// VisionSensors/Balluff BVS/fbBvsControl_ComIO
FUNCTION_BLOCK fbBvsControl_ComIO IMPLEMENTS I_VisionSensorSTD
VAR_IN_OUT
	stIO_Data: stVisionSensor_DigInOut;
END_VAR
VAR_INPUT
	bTrigger:BOOL;
	bReadActualInspection:BOOL;
	bChangeInspection:BOOL;		// Zbocze narastające inicjuje zmianę programu
	iInspectionToActive:INT;
	tMinImpWidth:TIME;		// Czas minimalnego trwania impulsu
END_VAR
VAR_OUTPUT
	bBusy: BOOL;
	bOutput1: BOOL;
	bOutput2: BOOL;
	bOutput3: BOOL;
	bError:	BOOL;
	bResultReady: BOOL;
	iActiveProgramId:INT;
END_VAR
VAR
	iWorkStep:INT;
	fbTP_ImpuleGen:TP;
	iImpulseToGenerate:INT;
	wConfirmedDeterctionNumber: WORD;
	fbTON_NewImpulsePause: TON;
	fbTON_Timeout: TON;
	bToggleMemory: BOOL;
	bNewInspectionBusy :BOOL;
	fbTON_CmdTimeout: TON;
	bReadInspectionBusy: BOOL;
	bSetInspectionBusy: BOOL;
	iIdToSet: INT;
	fbTON_NewStep: TON;
	fbTP_ImpulesRead: TP;
	fbTON_NewStepLong: TON;
	iTargetIdToSet: INT;
END_VAR

IF iWorkStep > 10 THEN
	fbTP_ImpuleGen(IN:= FALSE, PT:= tMinImpWidth + T#5MS);	
	fbTP_ImpulesRead(IN:= FALSE, PT:= 2*tMinImpWidth);	
	fbTON_NewStep(IN:= TRUE,PT:= tMinImpWidth);
	fbTON_NewStepLong(IN:= TRUE,PT:= 2*tMinImpWidth);
	IF iWorkStep < 90 THEN
		fbTON_CmdTimeout(IN:= TRUE, PT:= T#7S);
		IF fbTON_CmdTimeout.Q THEN
			fbTON_CmdTimeout(IN:= FALSE);
			iWorkStep := 90;
		END_IF
	END_IF	
END_IF


CASE iWorkStep OF
	0:	// Inicjalizacja
		IF bNewInspectionBusy OR bTrigger THEN		// Nowa detekcja
			bBusy := TRUE;
			bError := bSetInspectionBusy := bReadInspectionBusy := bOutput1 := bOutput2 := bOutput3 := bResultReady := FALSE;
			stIO_Data.bOut0_Trigger := TRUE;
			bToggleMemory:= stIO_Data.bIn0;
			fbTON_CmdTimeout(IN:= FALSE);
			iWorkStep := 10;
		ELSIF bReadInspectionBusy OR bReadActualInspection THEN		// Odczyt Id detekcji
			bBusy := TRUE;
			bError := bSetInspectionBusy := bResultReady := FALSE;
			iIdToSet := 21;
			iActiveProgramId := -1;
			fbTON_CmdTimeout(IN:= FALSE);
			iWorkStep := 20;
		ELSIF bSetInspectionBusy OR bChangeInspection THEN			// Ustawienie nowej detekcji
			IF bChangeInspection THEN
				IF iInspectionToActive > 0 AND iInspectionToActive <= 20 THEN
					iIdToSet := iInspectionToActive;
				END_IF		
			END_IF
			IF iIdToSet > 0 AND iIdToSet <= 20 THEN 			
				bBusy := TRUE;
				bError := bResultReady := FALSE;
				iTargetIdToSet:= iIdToSet;
				iActiveProgramId := -1;
				fbTON_CmdTimeout(IN:= FALSE);
				iWorkStep := 20;
			ELSE	
				bBusy := FALSE;
				bError := bResultReady := TRUE;
				iActiveProgramId := -1;
				iWorkStep := 1;
			END_IF
		END_IF
		
	1:	// Oczekiwanie po wykonanej komendzie na sygnał zerowy na poszczególnych wejściach
		IF NOT bTrigger AND NOT bReadActualInspection AND NOT bChangeInspection THEN
			fbTON_CmdTimeout(IN:= TRUE, PT:= T#1S);
			IF (NOT bNewInspectionBusy AND NOT bReadInspectionBusy AND NOT bSetInspectionBusy) OR fbTON_CmdTimeout.Q THEN
				bNewInspectionBusy := bReadInspectionBusy := bSetInspectionBusy := FALSE;
				bBusy := stIO_Data.bOut0_Trigger := stIO_Data.bOut1 := FALSE;
				fbTON_CmdTimeout(IN:= FALSE);
				iWorkStep := 0;
			END_IF	
		END_IF
	
	10:	// Detekcja wyzwolona, oczekiwanie na rezultat
		fbTON_CmdTimeout(IN:= TRUE, PT:= T#500MS);
		IF bToggleMemory <> stIO_Data.bIn0 THEN		// Detekcja zakończona
			bOutput1 := stIO_Data.bIn1;
			bOutput2 := stIO_Data.bInOut2;
			bOutput3 := stIO_Data.bInOut3;
			bResultReady := TRUE;
			bBusy := FALSE;
			bToggleMemory := stIO_Data.bIn0;
			stIO_Data.bOut0_Trigger := FALSE;
			iWorkStep := 1;
		ELSIF fbTON_CmdTimeout.Q THEN
			bBusy := FALSE;
			bError := TRUE;
			fbTON_CmdTimeout(IN:= FALSE);
			stIO_Data.bOut0_Trigger := FALSE;
			iWorkStep := 1;
		END_IF
		IF iWorkStep <> 10 THEN fbTON_CmdTimeout(IN:= FALSE); END_IF
				
		
	20:	// Odczyt/zmiana aktywnego programu 
		stIO_Data.bOut0_Trigger := stIO_Data.bOut1 := FALSE;
		fbTON_NewStep(IN:= FALSE);
		iWorkStep := 21;
	21:	// ***** FAZA 1 ***** Ustawienie sygnału wyboru programu	
		IF fbTON_NewStep.Q THEN
			stIO_Data.bOut1 := TRUE;
			fbTON_NewStep(IN:= FALSE);
			iWorkStep := 22;
		END_IF	
	22:	// ***** FAZA 2 ***** Oczekiwanie na wygaszenie wyjść i generacja impulsu
		IF NOT stIO_Data.bIn1 AND NOT stIO_Data.bInOut2 AND NOT stIO_Data.bInOut3 AND fbTON_NewStep.Q THEN
			fbTP_ImpuleGen(IN:= NOT stIO_Data.bOut0_Trigger);
			stIO_Data.bOut0_Trigger := fbTP_ImpuleGen.Q;
			iWorkStep := 23;	
		END_IF
	23:
		stIO_Data.bOut0_Trigger := fbTP_ImpuleGen.Q;
		IF NOT stIO_Data.bOut0_Trigger THEN
			fbTON_NewStep(IN:= FALSE);
			iWorkStep := 24;	
		END_IF	
	24:	// ***** FAZA 3 ***** Oczekiwanie na wystawienie wyjść
		IF stIO_Data.bIn1 AND stIO_Data.bInOut2 AND stIO_Data.bInOut3 AND fbTON_NewStep.Q THEN
			fbTON_NewStep(IN:= FALSE);
			iWorkStep := 25;	
		END_IF
	25:	// ***** FAZA 3 ***** Generacja liczby impulsów odpowiadających numerowi detekcji
		IF iIdToSet > 0 THEN
			iWorkStep := 26;
		ELSE
			fbTON_NewStep(IN:= FALSE);
			iWorkStep := 27;
		END_IF
	26:	// ***** FAZA 3 ***** Generacja liczby impulsów odpowiadających numerowi detekcji
		fbTP_ImpuleGen(IN:= NOT stIO_Data.bOut0_Trigger);
		stIO_Data.bOut0_Trigger := fbTP_ImpuleGen.Q;
		IF NOT stIO_Data.bOut0_Trigger THEN
			iIdToSet := iIdToSet -1;
			fbTON_NewStep(IN:= FALSE);
			iWorkStep := 27;
		END_IF
	27:	// ***** FAZA 3 ***** Pauza pomiędzy impulsami
		IF fbTON_NewStep.Q THEN
			IF iIdToSet > 0 THEN
				iWorkStep := 25;
			ELSE
				iWorkStep := 28;
			END_IF
		END_IF
	28:	// ***** FAZA 4 ***** Kasowanie sygnału ustawienia inspekcji
		stIO_Data.bOut0_Trigger := stIO_Data.bOut1 := FALSE;
		IF NOT stIO_Data.bIn1 AND NOT stIO_Data.bInOut2 AND NOT stIO_Data.bInOut3 THEN
			fbTON_NewStep(IN:= FALSE);
			iWorkStep := 29;
		END_IF
	29:	// Wystawienie pierwszego sygnału trigger
		IF fbTON_NewStep.Q THEN
			fbTP_ImpulesRead(IN:= NOT stIO_Data.bOut0_Trigger);
			stIO_Data.bOut0_Trigger := fbTP_ImpulesRead.Q;
			IF NOT stIO_Data.bOut0_Trigger THEN
				wConfirmedDeterctionNumber.0 := stIO_Data.bIn1;
				wConfirmedDeterctionNumber.1 := stIO_Data.bInOut2;
				wConfirmedDeterctionNumber.2 := stIO_Data.bInOut3;
				fbTON_NewStepLong(IN:= FALSE);
				iWorkStep := 30;
			END_IF
		END_IF
		
	30:
		IF NOT stIO_Data.bIn1 AND NOT stIO_Data.bInOut2 AND NOT stIO_Data.bInOut3 AND fbTON_NewStepLong.Q THEN
			fbTON_NewStep(IN:= FALSE);
			iWorkStep := 31;
		END_IF
	31:
		IF fbTON_NewStep.Q THEN
			fbTP_ImpulesRead(IN:= NOT stIO_Data.bOut0_Trigger);
			stIO_Data.bOut0_Trigger := fbTP_ImpulesRead.Q;
			IF NOT stIO_Data.bOut0_Trigger THEN
				wConfirmedDeterctionNumber.3 := stIO_Data.bIn1;
				wConfirmedDeterctionNumber.4 := stIO_Data.bInOut2;
				wConfirmedDeterctionNumber.5 := stIO_Data.bInOut3;
				fbTON_NewStepLong(IN:= FALSE);
				iWorkStep := 32;
			END_IF
		END_IF
	32:
		IF NOT stIO_Data.bIn1 AND NOT stIO_Data.bInOut2 AND NOT stIO_Data.bInOut3 AND fbTON_NewStepLong.Q THEN
			fbTON_NewStep(IN:= FALSE);
			iWorkStep := 33;
		END_IF
	33:
		IF fbTON_NewStep.Q THEN
			fbTP_ImpuleGen(IN:= NOT stIO_Data.bOut0_Trigger);
			stIO_Data.bOut0_Trigger := fbTP_ImpuleGen.Q;
			IF NOT stIO_Data.bOut0_Trigger THEN
				iWorkStep := 34;
			END_IF
		END_IF
	34:
		IF NOT stIO_Data.bIn1 AND NOT stIO_Data.bInOut2 AND NOT stIO_Data.bInOut3 THEN
			bBusy := FALSE;
			iActiveProgramId := WORD_TO_INT(wConfirmedDeterctionNumber);
			bResultReady := TRUE;
			bError := iTargetIdToSet = iActiveProgramId;
			iWorkStep := 1;
		END_IF
			
	90:	// In case of error ...
		bError := TRUE;
		bBusy := FALSE;
		stIO_Data.bOut0_Trigger := stIO_Data.bOut1 := FALSE;
		fbTON_CmdTimeout(IN:= TRUE, PT:= T#2S);
		IF fbTON_CmdTimeout.Q THEN
			iWorkStep := 1; 
		END_IF

END_CASE

METHOD mNewInspection : BOOL (* Metoda zwraca true gdy detekcja zostanie zakończona*)
VAR_OUTPUT
	bError	: BOOL;			// Informacja zakończeniu detekcji z błędem
	bOut1, bOut2, bOut3, bOut4	: BOOL;		// Wyjścia zostają odświeżone po zakońcoznej detekcji 
END_VAR
IF iWorkStep = 0 THEN
	bOut1 := bOut2 := bOut3 := bOut1 := bResultReady := FALSE;
	bNewInspectionBusy := TRUE;
ELSIF bNewInspectionBusy THEN
	IF bResultReady THEN
		bOut1 := bOutput1;
		bOut2 := bOutput2;
		bOut3 := bOutput3;
		bNewInspectionBusy := bError := bOut4 := FALSE;
		mNewInspection := TRUE;
	ELSIF fbTON_CmdTimeout.Q THEN
		bError := mNewInspection := TRUE;	
		bNewInspectionBusy := FALSE;
	END_IF
ELSE
	bError := mNewInspection := TRUE;
END_IF
END_METHOD

METHOD mReadInspectionId : BOOL (* Metoda zwraca true gdy zakończyła pracę*)
VAR_OUTPUT
	bError	: BOOL;			// Błąd ustawienia
	iActiveInspectionId	: INT;		// Identyfikator aktualnej inspekcji
END_VAR
IF iWorkStep = 0 THEN
	bResultReady := FALSE;
	bReadInspectionBusy := TRUE;
ELSIF bReadInspectionBusy THEN
	IF bResultReady THEN
		bReadInspectionBusy := bError := FALSE;
		iActiveInspectionId := iActiveProgramId;
		mReadInspectionId := TRUE;
	ELSIF fbTON_CmdTimeout.Q THEN
		bError := mReadInspectionId := TRUE;	
		iActiveInspectionId := -1;
		bReadInspectionBusy := FALSE;
	END_IF
ELSE
	bError := mReadInspectionId := TRUE;
	iActiveInspectionId := -1;
END_IF
END_METHOD

METHOD mSetInspectionId : BOOL
VAR_OUTPUT
	bError	: BOOL; 		// Błąd ustawienia
	iActiveInspectionId	: INT;		// Identyfikator aktualnej inspekcji
END_VAR
VAR_INPUT
	iInspectionIdToSet	: INT;			// Identyfikator inspekcji do ustawienia
END_VAR
IF iWorkStep = 0 AND iInspectionIdToSet <= 20 AND iInspectionIdToSet > 0 THEN
	bResultReady := FALSE;
	iIdToSet := iInspectionIdToSet;
	bSetInspectionBusy := TRUE;
ELSIF bSetInspectionBusy THEN
	IF bResultReady THEN
		bSetInspectionBusy := bError := FALSE;
		bError := iActiveProgramId <> iInspectionIdToSet;
		iActiveInspectionId := iActiveProgramId;
		mSetInspectionId := TRUE;
	ELSIF fbTON_CmdTimeout.Q THEN
		bError := mSetInspectionId := TRUE;	
		iActiveInspectionId := -1;
		bSetInspectionBusy := FALSE;
	END_IF
ELSE
	bError := mSetInspectionId := TRUE;
	iActiveInspectionId := -1;
END_IF
END_METHOD

END_FUNCTION_BLOCK

// VisionSensors/Cognex/fbCognexIS280Control
FUNCTION_BLOCK fbCognexIS280Control IMPLEMENTS I_VisionSensorSTD
VAR_IN_OUT
	stIO_Data: stCognexIS280_DigInOut;
END_VAR
VAR_INPUT
	bTrigger:BOOL;
	bReadActualInspection:BOOL;
	bChangeInspection:BOOL;		// Zbocze narastające inicjuje zmianę programu
	iInspectionToActive:INT;
	tMinImpWidth:TIME;		// Czas minimalnego trwania impulsu
END_VAR
VAR_OUTPUT
	bBusy: BOOL;
	bOutput1: BOOL;
	bOutput2: BOOL;
	bOutput3: BOOL;
	bError:	BOOL;
	bResultReady: BOOL;
	iActiveProgramId:INT;
END_VAR
VAR
	iWorkStep:INT;
	fbTP_ImpuleGen:TP;
	fbTON_Timeout: TON;
	bNewInspectionBusy :BOOL;
	fbTON_CmdTimeout: TON;
	iIdToSet: INT;
	fbTON_NewStep: TON;
	fbTP_ImpulesRead: TP;
	fbTON_NewStepLong: TON;
	iTargetIdToSet: INT;
END_VAR


CASE iWorkStep OF
	0:	// Inicjalizacja
		IF bNewInspectionBusy OR bTrigger THEN		// Nowa detekcja
			bBusy := TRUE;
		//	bSetInspectionBusy := bReadInspectionBusy := FALSE;
			bError := bOutput1 := bOutput2 := bOutput3 := bResultReady := FALSE;
			stIO_Data.bOut0_Trigger := TRUE;
			fbTON_CmdTimeout(IN:= FALSE);
			iWorkStep := 10;
		(*ELSIF bReadInspectionBusy OR bReadActualInspection THEN		// Odczyt Id detekcji
			bBusy := TRUE;
			bError := bSetInspectionBusy := bResultReady := FALSE;
			iIdToSet := 21;
			iActiveProgramId := -1;
			fbTON_CmdTimeout(IN:= FALSE);
			iWorkStep := 20;
		ELSIF bSetInspectionBusy OR bChangeInspection THEN			// Ustawienie nowej detekcji
			IF bChangeInspection THEN
				IF iInspectionToActive > 0 AND iInspectionToActive <= 20 THEN
					iIdToSet := iInspectionToActive;
				END_IF		
			END_IF
			IF iIdToSet > 0 AND iIdToSet <= 20 THEN 			
				bBusy := TRUE;
				bError := bResultReady := FALSE;
				iTargetIdToSet:= iIdToSet;
				iActiveProgramId := -1;
				fbTON_CmdTimeout(IN:= FALSE);
				iWorkStep := 20;
			ELSE	
				bBusy := FALSE;
				bError := bResultReady := TRUE;
				iActiveProgramId := -1;
				iWorkStep := 1;
			END_IF*)
		END_IF
		
	1:	// Oczekiwanie po wykonanej komendzie na sygnał zerowy na poszczególnych wejściach
		IF NOT bTrigger AND NOT bReadActualInspection AND NOT bChangeInspection THEN
			fbTON_CmdTimeout(IN:= TRUE, PT:= T#1S);
			IF NOT bNewInspectionBusy OR fbTON_CmdTimeout.Q THEN
				bNewInspectionBusy := FALSE;
				bBusy := stIO_Data.bOut0_Trigger := stIO_Data.bOut1 := FALSE;
				fbTON_CmdTimeout(IN:= FALSE);
				iWorkStep := 0;
			END_IF
		END_IF
	
	10:	// Detekcja wyzwolona, oczekiwanie na rezultat
		fbTON_CmdTimeout(IN:= TRUE, PT:= T#100MS);
		IF stIO_Data.bIn0 THEN
			iWorkStep := 11;
		ELSIF fbTON_CmdTimeout.Q THEN
			bBusy := FALSE;
			bError := TRUE;
			fbTON_CmdTimeout(IN:= FALSE);
			stIO_Data.bOut0_Trigger := FALSE;
			iWorkStep := 1;
		END_IF
		
	11:	// Oczekiwanie na koniec
		fbTON_CmdTimeout(IN:= TRUE, PT:= T#600MS);
		IF NOT stIO_Data.bIn0 THEN		// Detekcja zakończona
			bOutput1 := stIO_Data.bIn1;
			bOutput2 := stIO_Data.bInOut2;
			bOutput3 := stIO_Data.bInOut3;
			bResultReady := TRUE;
			bBusy := FALSE;
			stIO_Data.bOut0_Trigger := FALSE;
			iWorkStep := 1;
		ELSIF fbTON_CmdTimeout.Q THEN
			bBusy := FALSE;
			bError := TRUE;
			fbTON_CmdTimeout(IN:= FALSE);
			stIO_Data.bOut0_Trigger := FALSE;
			iWorkStep := 1;
		END_IF
				
	90:	// In case of error ...
		bError := TRUE;
		bBusy := FALSE;
		stIO_Data.bOut0_Trigger := stIO_Data.bOut1 := FALSE;
		fbTON_CmdTimeout(IN:= TRUE, PT:= T#2S);
		IF fbTON_CmdTimeout.Q THEN
			iWorkStep := 1; 
		END_IF

END_CASE

METHOD mNewInspection : BOOL (* Metoda zwraca true gdy detekcja zostanie zakończona*)
VAR_OUTPUT
	bError	: BOOL;			// Informacja zakończeniu detekcji z błędem
	bOut1, bOut2, bOut3, bOut4	: BOOL;		// Wyjścia zostają odświeżone po zakońcoznej detekcji 
END_VAR
IF iWorkStep = 0 THEN
	bOut1 := bOut2 := bOut3 := bOut1 := bResultReady := FALSE;
	bNewInspectionBusy := TRUE;
ELSIF bNewInspectionBusy THEN
	IF bResultReady THEN
		bOut1 := bOutput1;
		bOut2 := bOutput2;
		bOut3 := bOutput3;
		bNewInspectionBusy := bError := bOut4 := FALSE;
		mNewInspection := TRUE;
	ELSIF fbTON_CmdTimeout.Q THEN
		bError := mNewInspection := TRUE;	
		bNewInspectionBusy := FALSE;
	END_IF
ELSE
	bError := mNewInspection := TRUE;
END_IF
END_METHOD

METHOD mReadInspectionId : BOOL (* Metoda zwraca true gdy zakończyła pracę*)
VAR_OUTPUT
	bError	: BOOL;			// Błąd ustawienia
	iActiveInspectionId	: INT;		// Identyfikator aktualnej inspekcji
END_VAR
bError :=  mReadInspectionId := TRUE;
iActiveInspectionId := -1;
(*IF iWorkStep = 0 THEN
	bResultReady := FALSE;
	bReadInspectionBusy := TRUE;
ELSIF bReadInspectionBusy THEN
	IF bResultReady THEN
		bReadInspectionBusy := bError := FALSE;
		iActiveInspectionId := iActiveProgramId;
		mReadInspectionId := TRUE;
	ELSIF fbTON_CmdTimeout.Q THEN
		bError := mReadInspectionId := TRUE;	
		iActiveInspectionId := -1;
		bReadInspectionBusy := FALSE;
	END_IF
ELSE
	bError := mReadInspectionId := TRUE;
	iActiveInspectionId := -1;
END_IF
*)
END_METHOD

METHOD mSetInspectionId : BOOL
VAR_OUTPUT
	bError	: BOOL; 		// Błąd ustawienia
	iActiveInspectionId	: INT;		// Identyfikator aktualnej inspekcji
END_VAR
VAR_INPUT
	iInspectionIdToSet	: INT;			// Identyfikator inspekcji do ustawienia
END_VAR
bError :=  mSetInspectionId := TRUE;
iActiveInspectionId := -1;

(*IF iWorkStep = 0 AND iInspectionIdToSet <= 20 AND iInspectionIdToSet > 0 THEN
	bResultReady := FALSE;
	iIdToSet := iInspectionIdToSet;
	bSetInspectionBusy := TRUE;
ELSIF bSetInspectionBusy THEN
	IF bResultReady THEN
		bSetInspectionBusy := bError := FALSE;
		bError := iActiveProgramId <> iInspectionIdToSet;
		iActiveInspectionId := iActiveProgramId;
		mSetInspectionId := TRUE;
	ELSIF fbTON_CmdTimeout.Q THEN
		bError := mSetInspectionId := TRUE;	
		iActiveInspectionId := -1;
		bSetInspectionBusy := FALSE;
	END_IF
ELSE
	bError := mSetInspectionId := TRUE;
	iActiveInspectionId := -1;
END_IF
*)
END_METHOD

END_FUNCTION_BLOCK

// VisionSensors/Keyence/fbKeyenceIVControl
FUNCTION_BLOCK fbKeyenceIVControl IMPLEMENTS I_VisionSensorSTD
VAR_IN_OUT
	stIO_Data: stKeyence_DigInOut;
END_VAR
VAR_INPUT
	bTrigger:BOOL;
	bReadActualInspection:BOOL;
	bChangeInspection:BOOL;		// Zbocze narastające inicjuje zmianę programu
	iInspectionToActive:INT;
	tMinImpWidth:TIME;		// Czas minimalnego trwania impulsu
END_VAR
VAR_OUTPUT
	bBusy: BOOL;
	bOutput1: BOOL;
	bOutput2: BOOL;
	bOutput3: BOOL;
	bError:	BOOL;
	bResultReady: BOOL;
	iActiveProgramId:INT;
END_VAR
VAR
	iWorkStep:INT;
	fbTP_ImpuleGen:TP;
	fbTON_Timeout: TON;
	bNewInspectionBusy, bSetInspectionBusy, bReadInspectionBusy :BOOL;
	fbTON_CmdTimeout: TON;
	iIdToSet: INT;
	fbTON_NewStep: TON;
	fbTP_ImpulesRead: TP;
	fbTON_NewStepLong: TON;
	iTargetIdToSet: INT;
END_VAR


CASE iWorkStep OF
	0:	// Inicjalizacja
		IF bNewInspectionBusy OR bTrigger THEN		// Nowa detekcja
			bBusy := TRUE;
		//	bSetInspectionBusy := bReadInspectionBusy := FALSE;
			bError := bOutput1 := bOutput2 := bOutput3 := bResultReady := FALSE;
			stIO_Data.bDO_IN1_Trigger := TRUE;
			fbTON_CmdTimeout(IN:= FALSE);
			iWorkStep := 10;
(*		ELSIF bReadInspectionBusy OR bReadActualInspection THEN		// Odczyt Id detekcji
			bBusy := TRUE;
			bError := bSetInspectionBusy := bResultReady := FALSE;
			iIdToSet := 21;
			iActiveProgramId := -1;
			fbTON_CmdTimeout(IN:= FALSE);
			iWorkStep := 20;
		ELSIF bSetInspectionBusy OR bChangeInspection THEN			// Ustawienie nowej detekcji
			IF bChangeInspection THEN
				IF iInspectionToActive > 0 AND iInspectionToActive <= 20 THEN
					iIdToSet := iInspectionToActive;
				END_IF		
			END_IF
			IF iIdToSet > 0 AND iIdToSet <= 20 THEN 			
				bBusy := TRUE;
				bError := bResultReady := FALSE;
				iTargetIdToSet:= iIdToSet;
				iActiveProgramId := -1;
				fbTON_CmdTimeout(IN:= FALSE);
				iWorkStep := 20;
			ELSE	
				bBusy := FALSE;
				bError := bResultReady := TRUE;
				iActiveProgramId := -1;
				iWorkStep := 1;
			END_IF	*)
		END_IF
		
	1:	// Oczekiwanie po wykonanej komendzie na sygnał zerowy na poszczególnych wejściach
		IF NOT bTrigger AND NOT bReadActualInspection AND NOT bChangeInspection THEN
			fbTON_CmdTimeout(IN:= TRUE, PT:= T#1S);
			IF NOT bNewInspectionBusy OR fbTON_CmdTimeout.Q THEN
				bNewInspectionBusy := FALSE;
				bBusy := stIO_Data.bDO_IN1_Trigger := FALSE;
				fbTON_CmdTimeout(IN:= FALSE);
				iWorkStep := 0;
			END_IF
		END_IF
	
	10:	// Detekcja wyzwolona, oczekiwanie na rezultat
		fbTON_CmdTimeout(IN:= TRUE, PT:= T#100MS);
		IF stIO_Data.bDI_OUT1_Busy THEN
			stIO_Data.bDO_IN1_Trigger := FALSE;
			iWorkStep := 11;
		ELSIF fbTON_CmdTimeout.Q THEN
			bBusy := FALSE;
			bError := TRUE;
			fbTON_CmdTimeout(IN:= FALSE);
			stIO_Data.bDO_IN1_Trigger := FALSE;
			iWorkStep := 1;
		END_IF
		
	11:	// Oczekiwanie na koniec
		fbTON_CmdTimeout(IN:= TRUE, PT:= T#600MS);
		IF NOT stIO_Data.bDI_OUT1_Busy THEN		// Detekcja zakończona
			bOutput1 := stIO_Data.bDI_OUT2;
			bOutput2 := stIO_Data.bDI_OUT3;
			bOutput3 := stIO_Data.bDI_OUT4;
			bResultReady := TRUE;
			bBusy := FALSE;
			stIO_Data.bDO_IN1_Trigger := FALSE;
			iWorkStep := 1;
		ELSIF fbTON_CmdTimeout.Q THEN
			bBusy := FALSE;
			bError := TRUE;
			fbTON_CmdTimeout(IN:= FALSE);
			stIO_Data.bDO_IN1_Trigger := FALSE;
			iWorkStep := 1;
		END_IF
				
	90:	// In case of error ...
		bError := TRUE;
		bBusy := FALSE;
		stIO_Data.bDO_IN1_Trigger := FALSE;
		fbTON_CmdTimeout(IN:= TRUE, PT:= T#2S);
		IF fbTON_CmdTimeout.Q THEN
			iWorkStep := 1; 
		END_IF

END_CASE

METHOD mNewInspection : BOOL (* Metoda zwraca true gdy detekcja zostanie zakończona*)
VAR_OUTPUT
	bError	: BOOL;			// Informacja zakończeniu detekcji z błędem
	bOut1, bOut2, bOut3, bOut4	: BOOL;		// Wyjścia zostają odświeżone po zakońcoznej detekcji 
END_VAR
IF iWorkStep = 0 THEN
	bOut1 := bOut2 := bOut3 := bOut1 := bResultReady := FALSE;
	bNewInspectionBusy := TRUE;
ELSIF bNewInspectionBusy THEN
	IF bResultReady THEN
		bOut1 := bOutput1;
		bOut2 := bOutput2;
		bOut3 := bOutput3;
		bNewInspectionBusy := bError := bOut4 := FALSE;
		mNewInspection := TRUE;
	ELSIF fbTON_CmdTimeout.Q THEN
		bError := mNewInspection := TRUE;	
		bNewInspectionBusy := FALSE;
	END_IF
ELSE
	bError := mNewInspection := TRUE;
END_IF
END_METHOD

METHOD mReadInspectionId : BOOL (* Metoda zwraca true gdy zakończyła pracę*)
VAR_OUTPUT
	bError	: BOOL;			// Błąd ustawienia
	iActiveInspectionId	: INT;		// Identyfikator aktualnej inspekcji
END_VAR
bError :=  mReadInspectionId := TRUE;
iActiveInspectionId := -1;
(*IF iWorkStep = 0 THEN
	bResultReady := FALSE;
	bReadInspectionBusy := TRUE;
ELSIF bReadInspectionBusy THEN
	IF bResultReady THEN
		bReadInspectionBusy := bError := FALSE;
		iActiveInspectionId := iActiveProgramId;
		mReadInspectionId := TRUE;
	ELSIF fbTON_CmdTimeout.Q THEN
		bError := mReadInspectionId := TRUE;	
		iActiveInspectionId := -1;
		bReadInspectionBusy := FALSE;
	END_IF
ELSE
	bError := mReadInspectionId := TRUE;
	iActiveInspectionId := -1;
END_IF
*)
END_METHOD

METHOD mSetInspectionId : BOOL
VAR_OUTPUT
	bError	: BOOL; 		// Błąd ustawienia
	iActiveInspectionId	: INT;		// Identyfikator aktualnej inspekcji
END_VAR
VAR_INPUT
	iInspectionIdToSet	: INT;			// Identyfikator inspekcji do ustawienia
END_VAR
bError :=  mSetInspectionId := TRUE;
iActiveInspectionId := -1;

(*IF iWorkStep = 0 AND iInspectionIdToSet <= 20 AND iInspectionIdToSet > 0 THEN
	bResultReady := FALSE;
	iIdToSet := iInspectionIdToSet;
	bSetInspectionBusy := TRUE;
ELSIF bSetInspectionBusy THEN
	IF bResultReady THEN
		bSetInspectionBusy := bError := FALSE;
		bError := iActiveProgramId <> iInspectionIdToSet;
		iActiveInspectionId := iActiveProgramId;
		mSetInspectionId := TRUE;
	ELSIF fbTON_CmdTimeout.Q THEN
		bError := mSetInspectionId := TRUE;	
		iActiveInspectionId := -1;
		bSetInspectionBusy := FALSE;
	END_IF
ELSE
	bError := mSetInspectionId := TRUE;
	iActiveInspectionId := -1;
END_IF
*)
END_METHOD

END_FUNCTION_BLOCK

// VisionSensors/Keyence/fbKeyenceIVControl_ComIO
FUNCTION_BLOCK fbKeyenceIVControl_ComIO IMPLEMENTS I_VisionSensorSTD
VAR_IN_OUT
	stIO_Data: stVisionSensor_DigInOut;
END_VAR
VAR_INPUT
	bTrigger:BOOL;
	bReadActualInspection:BOOL;
	bChangeInspection:BOOL;		// Zbocze narastające inicjuje zmianę programu
	iInspectionToActive:INT;
	tMinImpWidth:TIME;		// Czas minimalnego trwania impulsu
END_VAR
VAR_OUTPUT
	bBusy: BOOL;
	bOutput1: BOOL;
	bOutput2: BOOL;
	bOutput3: BOOL;
	bError:	BOOL;
	bResultReady: BOOL;
	iActiveProgramId:INT;
END_VAR
VAR
	iWorkStep:INT;
	fbTP_ImpuleGen:TP;
	fbTON_Timeout: TON;
	bNewInspectionBusy, bSetInspectionBusy, bReadInspectionBusy :BOOL;
	fbTON_CmdTimeout: TON;
	iIdToSet: INT;
	fbTON_NewStep: TON;
	fbTP_ImpulesRead: TP;
	fbTON_NewStepLong: TON;
	iActInspectionId: INT;
END_VAR


CASE iWorkStep OF
	0:	// Inicjalizacja
		IF bNewInspectionBusy OR bTrigger THEN		// Nowa detekcja
			bBusy := TRUE;
		//	bSetInspectionBusy := bReadInspectionBusy := FALSE;
			bError := bOutput1 := bOutput2 := bOutput3 := bResultReady := FALSE;
			stIO_Data.bOut0_Trigger := TRUE;
			fbTON_CmdTimeout(IN:= FALSE);
			iWorkStep := 10;
		ELSIF bReadInspectionBusy OR bReadActualInspection THEN		// Odczyt Id detekcji
			bBusy := TRUE;
			iActiveProgramId := 0;
			iActiveProgramId.0 := stIO_Data.bOut1;
			iActiveProgramId.1 := stIO_Data.bOut2;
			iActiveProgramId.2 := stIO_Data.bOut3;
			iActiveProgramId.3 := stIO_Data.bOut4;
			bError := bSetInspectionBusy := FALSE;
			fbTON_CmdTimeout(IN:= FALSE);
			bError := bBusy := FALSE;
			bResultReady := TRUE;
			iWorkStep := 1;
			
		ELSIF bSetInspectionBusy OR bChangeInspection THEN			// Ustawienie nowej detekcji
			IF bChangeInspection THEN
				IF iInspectionToActive > 0 AND iInspectionToActive <= 15 THEN
					iIdToSet := iInspectionToActive;
				END_IF		
			END_IF
			IF iIdToSet > 0 AND iIdToSet <= 15 THEN 			
				bBusy := TRUE;
				stIO_Data.bOut1 := iIdToSet.0;
				stIO_Data.bOut2 := iIdToSet.1;
				stIO_Data.bOut3 := iIdToSet.2;
				stIO_Data.bOut4 := iIdToSet.3;
				iActiveProgramId := iIdToSet;
				bError := FALSE;
				bResultReady := TRUE;
				fbTON_CmdTimeout(IN:= FALSE);
				iWorkStep := 1;
			ELSE	
				bBusy := FALSE;
				bError := bResultReady := TRUE;
				iActiveProgramId := -1;
				iWorkStep := 1;
			END_IF	
		END_IF
		
	1:	// Oczekiwanie po wykonanej komendzie na sygnał zerowy na poszczególnych wejściach
		IF NOT bTrigger AND NOT bReadActualInspection AND NOT bChangeInspection THEN
			fbTON_CmdTimeout(IN:= TRUE, PT:= T#1S);
			IF NOT bNewInspectionBusy OR fbTON_CmdTimeout.Q THEN
				bNewInspectionBusy := FALSE;
				bBusy := stIO_Data.bOut0_Trigger := FALSE;
				fbTON_CmdTimeout(IN:= FALSE);
				iWorkStep := 0;
			END_IF
		END_IF
	
	10:	// Detekcja wyzwolona, oczekiwanie na rezultat
		fbTON_CmdTimeout(IN:= TRUE, PT:= T#100MS);
		IF stIO_Data.bIn0 THEN
			stIO_Data.bOut0_Trigger := FALSE;
			iWorkStep := 11;
		ELSIF fbTON_CmdTimeout.Q THEN
			bBusy := FALSE;
			bError := TRUE;
			fbTON_CmdTimeout(IN:= FALSE);
			stIO_Data.bOut0_Trigger := FALSE;
			iWorkStep := 1;
		END_IF
		
	11:	// Oczekiwanie na koniec
		fbTON_CmdTimeout(IN:= TRUE, PT:= T#600MS);
		IF NOT stIO_Data.bIn0 THEN		// Detekcja zakończona
			bOutput1 := stIO_Data.bIn1;
			bOutput2 := stIO_Data.bInOut2;
			bOutput3 := stIO_Data.bInOut3;
			bResultReady := TRUE;
			bBusy := FALSE;
			stIO_Data.bOut0_Trigger := FALSE;
			iWorkStep := 1;
		ELSIF fbTON_CmdTimeout.Q THEN
			bBusy := FALSE;
			bError := TRUE;
			fbTON_CmdTimeout(IN:= FALSE);
			stIO_Data.bOut0_Trigger := FALSE;
			iWorkStep := 1;
		END_IF
				
	90:	// In case of error ...
		bError := TRUE;
		bBusy := FALSE;
		stIO_Data.bOut0_Trigger := FALSE;
		fbTON_CmdTimeout(IN:= TRUE, PT:= T#2S);
		IF fbTON_CmdTimeout.Q THEN
			iWorkStep := 1; 
		END_IF

END_CASE

METHOD mNewInspection : BOOL (* Metoda zwraca true gdy detekcja zostanie zakończona*)
VAR_OUTPUT
	bError	: BOOL;			// Informacja zakończeniu detekcji z błędem
	bOut1, bOut2, bOut3, bOut4	: BOOL;		// Wyjścia zostają odświeżone po zakońcoznej detekcji 
END_VAR
IF iWorkStep = 0 THEN
	bOut1 := bOut2 := bOut3 := bOut1 := bResultReady := FALSE;
	bNewInspectionBusy := TRUE;
ELSIF bNewInspectionBusy THEN
	IF bResultReady THEN
		bOut1 := bOutput1;
		bOut2 := bOutput2;
		bOut3 := bOutput3;
		bNewInspectionBusy := bError := bOut4 := FALSE;
		mNewInspection := TRUE;
	ELSIF fbTON_CmdTimeout.Q THEN
		bError := mNewInspection := TRUE;	
		bNewInspectionBusy := FALSE;
	END_IF
ELSE
	bError := mNewInspection := TRUE;
END_IF
END_METHOD

METHOD mReadInspectionId : BOOL (* Metoda zwraca true gdy zakończyła pracę*)
VAR_OUTPUT
	bError	: BOOL;			// Błąd ustawienia
	iActiveInspectionId	: INT;		// Identyfikator aktualnej inspekcji
END_VAR
VAR
	
END_VAR
//mReadInspectionId := TRUE;

IF iWorkStep = 0 THEN
	bResultReady := FALSE;
	bReadInspectionBusy := TRUE;
	iActiveProgramId := -1;
ELSIF bReadInspectionBusy THEN
	IF bResultReady THEN
		bReadInspectionBusy := bError := FALSE;
		iActiveInspectionId := iActiveProgramId;
		mReadInspectionId := TRUE;
	ELSIF fbTON_CmdTimeout.Q THEN
		bError := mReadInspectionId := TRUE;	
		iActiveInspectionId := -1;
		bReadInspectionBusy := FALSE;
	END_IF
ELSE
	bError := mReadInspectionId := TRUE;
	iActiveInspectionId := -1;
END_IF
END_METHOD

METHOD mSetInspectionId : BOOL
VAR_OUTPUT
	bError	: BOOL; 		// Błąd ustawienia
	iActiveInspectionId	: INT;		// Identyfikator aktualnej inspekcji
END_VAR
VAR_INPUT
	iInspectionIdToSet	: INT;			// Identyfikator inspekcji do ustawienia
END_VAR
iActiveInspectionId := -1;
IF iWorkStep = 0 AND iInspectionIdToSet <= 15 AND iInspectionIdToSet > 0 THEN
	bResultReady := FALSE;
	iIdToSet := iInspectionIdToSet;
	bSetInspectionBusy := TRUE;
ELSIF bSetInspectionBusy THEN
	IF bResultReady THEN
		bSetInspectionBusy := bError := FALSE;
		bError S= iActiveProgramId <> iInspectionIdToSet;
		iActiveInspectionId := iActiveProgramId;
		mSetInspectionId := TRUE;
	ELSIF fbTON_CmdTimeout.Q THEN
		bError := mSetInspectionId := TRUE;	
		iActiveInspectionId := -1;
		bSetInspectionBusy := FALSE;
	END_IF
ELSE
	bError := mSetInspectionId := TRUE;
	iActiveInspectionId := -1;
END_IF
END_METHOD

END_FUNCTION_BLOCK

// ReadMe
PROGRAM ReadMe
VAR
(*	// SQL
	fbSQL: fbSQL_Core;
	
	// PIM
	fbPIM_Full: fbPIM_Station_V3;
	fbPIM_Simple: fbPIM_SimplePimStation;
	fbPIM_Dummy: fbPIM_Dummy;
	fbPIM_UsLogin: fbPIM_UserLogin;
	
	// Vision
	fbBalluff: fbBvsControl;
	fbKeyence: fbKeyenceIVControl;
	fbCognex: fbCognexIS280Control;
	
	// Loggers
	fbTextLogger: fbTextDataLogger;
	
	//Common
	fbAssemblyPos: fbAssemblyPost;
	fb2HaStart: fb2HandStart;
	fbActuator:fbActuator;
	fbActuatorOOP:fbActuatorOOP;
*)	
	
END_VAR


(*
Tipy:
Obsługa bibliotek- istnieje możliwość redefinicji lokalnej dla struktur i bloków z biblioteki. Jeśli chcemy użyć bloku z biblioteki dodajemy przedrostek z nazwą biblioteki w polu deklaracji znmiennej.
					Jeśli go nie dodamy wtedy TwinCAT użyje lokalnych plików

Teksty do wyświetlenia w kompilatorze:
					{text 'Tekst do wyświetlenia'}
					{info 'Tekst do wyświetlenia'}
					{warning 'Tekst do wyświetlenia'}
					{error 'Tekst do wyświetlenia'}



*)

END_PROGRAM

// Common/RecipeManager/VISUs/vRecipeManager_Ctrl
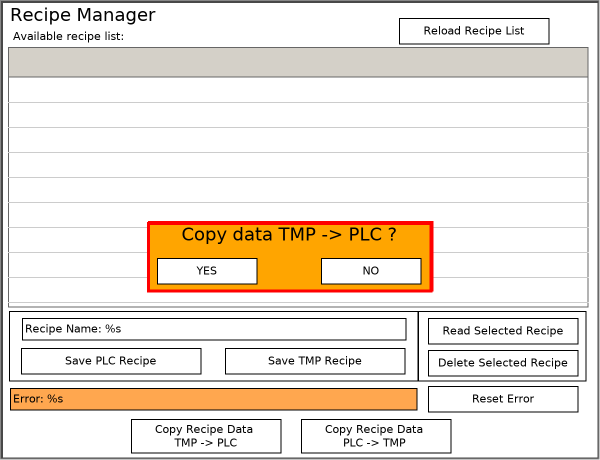
VISUALIZATION vRecipeManager_Ctrl  // 600x460
VAR_IN_OUT
	fbRecipe:fbRecipeManager;
END_VAR
    Rectangle (1,1 598x458)
    Rectangle (418,311 168x70)
    Rectangle (9,311 409x70)
    Table (8,47 580x260), data array: fbRecipe.astRecipeList
        p1128707560: fbRecipe.iNbOfFoundRecipes
        p1137915858: fbRecipe.iTableSelIndex
        p1822360349: fbRecipe.bTableRowSelected
        p3854506369: fbRecipe.astRecipeList[INDEX].sFileName
        p1892666644: fbRecipe.astRecipeList[INDEX].dtCreationTime
        p2232123230: Recipe Name
        p511219082: Creation Time
    Label (7,0 150x30), "Recipe Manager"
    Label (10,29 150x15), "Available recipe list:"
    RoundedRectangle (399,18 150x26), "Reload Recipe List", colour toggle: fbRecipe.bRefreshingRecipeList
        toggle fbRecipe.bReloadRecipes
    RoundedRectangle (21,348 180x26), "Save PLC Recipe", colour toggle: fbRecipe.bWritingRecipe
        OnMouseClick: execute { fbRecipe.bWriteRecipe := NOT fbRecipe.bWriteRecipe; fbRecipe.bSavePLCStruct := TRUE; }
    Rectangle (22,318 384x22), "Recipe Name: %s", text variable: fbRecipe.sRecipeName
        OnMouseClick: write fbRecipe.sRecipeName via Default, title 'New Recipe Name', format %s
    RoundedRectangle (131,419 150x34), "Copy Recipe Data TMP -> PLC", colour toggle: fbRecipe.bCopyTMP_2_PLC
        toggle fbRecipe.bCopyTMP_2_PLC
    RoundedRectangle (301,419 150x34), "Copy Recipe Data PLC -> TMP", colour toggle: fbRecipe.bCopyPLC_2_TMP
        toggle fbRecipe.bCopyPLC_2_TMP
    RoundedRectangle (428,318 150x26), "Read Selected Recipe", colour toggle: fbRecipe.bReadingRecipe
        toggle fbRecipe.bReadRecipe
    RoundedRectangle (225,348 180x26), "Save TMP Recipe", colour toggle: fbRecipe.bWritingRecipe
        OnMouseClick: execute { fbRecipe.bWriteRecipe := NOT fbRecipe.bWriteRecipe; fbRecipe.bSavePLCStruct := FALSE; }
    Rectangle (10,388 407x22), "Error: %s", text variable: fbRecipe.nErrorCode, invisible if: NOT fbRecipe.bError
        OnMouseClick: write fbRecipe.sRecipeName via Default, title 'New Recipe Name', format %s
    RoundedRectangle (428,386 150x26), "Reset Error", colour toggle: fbRecipe.bResetInternal, invisible if: NOT fbRecipe.bError
        toggle fbRecipe.bResetInternal
    RoundedRectangle (428,350 150x26), "Delete Selected Recipe", colour toggle: fbRecipe.bDeletingRecipe
        toggle fbRecipe.bDeleteRecipe
    Group (148,221 285x70), invisible if: NOT fbRecipe.bDeleteRecipe
        Rectangle (0,0 285x70), "Delete selection ?"
        RoundedRectangle (10,36 100x26), "YES"
            toggle fbRecipe.bDeleteConfirmed
        RoundedRectangle (174,36 100x26), "NO"
            toggle fbRecipe.bDeleteRecipe
    Group (147,222 285x70), invisible if: NOT fbRecipe.bCopyTMP_2_PLC
        Rectangle (0,0 285x70), "Copy data TMP -> PLC ?"
        RoundedRectangle (10,36 100x26), "YES"
            toggle fbRecipe.bCopyTMP_2_PLC_Confirmed
        RoundedRectangle (174,36 100x26), "NO"
            toggle fbRecipe.bCopyTMP_2_PLC
END_VISUALIZATION

// Common/RecipeManager/VISUs/vRecipeManager_CtrlWide
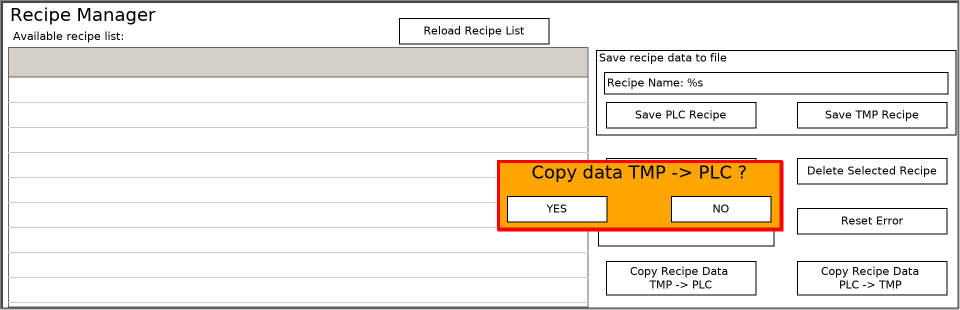
VISUALIZATION vRecipeManager_CtrlWide  // 960x310
VAR_IN_OUT
	fbRecipe:fbRecipeManager;
END_VAR
    Rectangle (1,1 958x308)
    Rectangle (596,50 360x85), "Save recipe data to file"
    Table (8,47 580x260), data array: fbRecipe.astRecipeList
        p1128707560: fbRecipe.iNbOfFoundRecipes
        p1137915858: fbRecipe.iTableSelIndex
        p1822360349: fbRecipe.bTableRowSelected
        p3854506369: fbRecipe.astRecipeList[INDEX].sFileName
        p1892666644: fbRecipe.astRecipeList[INDEX].dtCreationTime
        p2232123230: Recipe Name
        p511219082: Creation Time
    Label (7,0 150x30), "Recipe Manager"
    Label (10,29 150x15), "Available recipe list:"
    RoundedRectangle (399,18 150x26), "Reload Recipe List", colour toggle: fbRecipe.bRefreshingRecipeList
        toggle fbRecipe.bReloadRecipes
    RoundedRectangle (606,102 150x26), "Save PLC Recipe", colour toggle: fbRecipe.bWritingRecipe
        OnMouseClick: execute { fbRecipe.bWriteRecipe := NOT fbRecipe.bWriteRecipe; fbRecipe.bSavePLCStruct := TRUE; }
    Rectangle (604,72 344x22), "Recipe Name: %s", text variable: fbRecipe.sRecipeName
        OnMouseClick: write fbRecipe.sRecipeName via Default, title 'New Recipe Name', format %s
    RoundedRectangle (606,261 150x34), "Copy Recipe Data TMP -> PLC", colour toggle: fbRecipe.bCopyTMP_2_PLC
        toggle fbRecipe.bCopyTMP_2_PLC
    RoundedRectangle (797,261 150x34), "Copy Recipe Data PLC -> TMP", colour toggle: fbRecipe.bCopyPLC_2_TMP
        toggle fbRecipe.bCopyPLC_2_TMP
    RoundedRectangle (606,158 150x26), "Read Selected Recipe", colour toggle: fbRecipe.bReadingRecipe
        toggle fbRecipe.bReadRecipe
    RoundedRectangle (797,102 150x26), "Save TMP Recipe", colour toggle: fbRecipe.bWritingRecipe
        OnMouseClick: execute { fbRecipe.bWriteRecipe := NOT fbRecipe.bWriteRecipe; fbRecipe.bSavePLCStruct := FALSE; }
    Rectangle (598,196 176x50), "Error: %s", text variable: fbRecipe.nErrorCode, invisible if: NOT fbRecipe.bError
        OnMouseClick: write fbRecipe.sRecipeName via Default, title 'New Recipe Name', format %s
    RoundedRectangle (797,208 150x26), "Reset Error", colour toggle: fbRecipe.bResetInternal, invisible if: NOT fbRecipe.bError
        toggle fbRecipe.bResetInternal
    RoundedRectangle (797,158 150x26), "Delete Selected Recipe", colour toggle: fbRecipe.bDeletingRecipe
        toggle fbRecipe.bDeleteRecipe
    Group (498,161 285x70), invisible if: NOT fbRecipe.bDeleteRecipe
        Rectangle (0,0 285x70), "Delete selection ?"
        RoundedRectangle (10,36 100x26), "YES"
            toggle fbRecipe.bDeleteConfirmed
        RoundedRectangle (174,36 100x26), "NO"
            toggle fbRecipe.bDeleteRecipe
    Group (497,160 285x70), invisible if: NOT fbRecipe.bCopyTMP_2_PLC
        Rectangle (0,0 285x70), "Copy data TMP -> PLC ?"
        RoundedRectangle (10,36 100x26), "YES"
            toggle fbRecipe.bCopyTMP_2_PLC_Confirmed
        RoundedRectangle (174,36 100x26), "NO"
            toggle fbRecipe.bCopyTMP_2_PLC
END_VISUALIZATION

// ProdLineMachines/AssemblyPost/VISUs/vAssemblyPost_Main
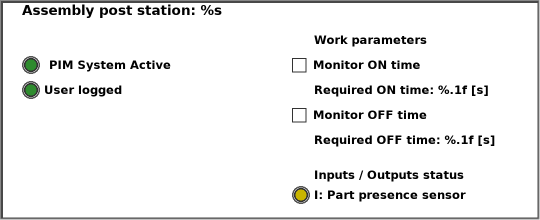
VISUALIZATION vAssemblyPost_Main  // 540x220
VAR_IN_OUT
	fbData:fbAssemblyPost;
END_VAR
    Rectangle (1,1 538x218), "Assembly post station: %s", text variable: fbData.stStationData.sNazwaStanowiska
    RoundedRectangle (18,55 193x20), "PIM System Active", colour toggle: NOT fbData.bPIM_Active
    Rectangle (311,80 200x20), "Required ON time: %.1f [s]", text variable: fbData.stWorkParams.rRequiredTimeON, input disabled if: NOT GVL.fbUserLogin.bPermissionGranted
        OnMouseClick: write the text variable via Default, min 0.5, max 30, title 'Required ON time', format %.1f
    Label (41,80 170x20), "User logged"
    Lamp1 (21,80 20x20), variable: fbData.bUserLogged, style: Lamp-Lamp1-Green
    Label (311,185 170x20), "I: Part presence sensor"
    Lamp1 (291,185 20x20), variable: fbData.fbPartFiltered.Q, style: Lamp-Lamp1-Yellow
    Label (311,165 170x20), "Inputs / Outputs status"
    Lamp1 (21,55 20x20), variable: fbData.bPIM_Active, style: Lamp-Lamp1-Green
    Rectangle (311,130 200x20), "Required OFF time: %.1f [s]", text variable: fbData.stWorkParams.rRequiredTimeOFF, input disabled if: NOT GVL.fbUserLogin.bPermissionGranted
        OnMouseClick: write the text variable via Default, min 0.5, max 30, title 'Required OFF time', format %.1f
    Checkbox (290,55 20x20), variable: fbData.stWorkParams.bMonitorON_Time, input disabled if: NOT GVL.fbUserLogin.bPermissionGranted
    Label (310,55 170x20), "Monitor ON time"
    Checkbox (290,105 20x20), variable: fbData.stWorkParams.bMonitorOFF_Time, input disabled if: NOT GVL.fbUserLogin.bPermissionGranted
    Label (310,105 170x20), "Monitor OFF time"
    Label (311,30 170x20), "Work parameters"
END_VISUALIZATION

// ProdLineMachines/Sonictech/Fixtures/S01_IndicatorAssembly/VISUs/SubFrame/vStFix_S01IndicatorAssy_SubDiag
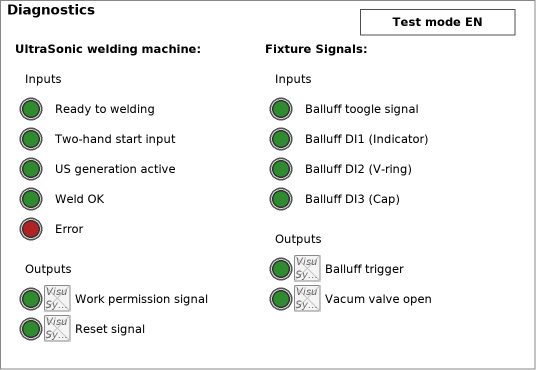
VISUALIZATION vStFix_S01IndicatorAssy_SubDiag  // 536x370
VAR_IN_OUT
	fbMachine: fbSonictechUSWM;
	stFixInOuts: stStFix_S01IndicatorAssy_InOut;
END_VAR
    Frame (0,0 536x370)
        shows vSonictechUSWM_SubDiag(fbMachine := fbMachine)
    Label (262,36 203x26), "Fixture Signals:"
    Rectangle (272,66 160x26), "Inputs"
    Lamp1 (268,96 26x26), variable: stFixInOuts.stBalluff.bDI_TriggerSignal, style: Lamp-Lamp1-Green
    Rectangle (302,96 160x26), "Balluff toogle signal"
    Lamp1 (268,126 26x26), variable: stFixInOuts.stBalluff.bDI_TriggerSignal, style: Lamp-Lamp1-Green
    Rectangle (302,126 160x26), "Balluff DI1 (Indicator)"
    Rectangle (302,156 160x26), "Balluff DI2 (V-ring)"
    Lamp1 (268,156 26x26), variable: stFixInOuts.stBalluff.bDI_TriggerSignal, style: Lamp-Lamp1-Green
    Lamp1 (268,186 26x26), variable: stFixInOuts.stBalluff.bDI_Input_3, style: Lamp-Lamp1-Green
    Rectangle (302,186 160x26), "Balluff DI3 (Cap)"
    Rectangle (272,226 160x26), "Outputs"
    Lamp1 (268,256 26x26), variable: stFixInOuts.stBalluff.bDO_Trigger, style: Lamp-Lamp1-Green
    Rectangle (322,256 150x26), "Balluff trigger"
    Lamp1 (268,286 26x26), variable: stFixInOuts.bVacuumON_Q, style: Lamp-Lamp1-Green
    Rectangle (322,286 150x26), "Vacum valve open"
    Image (294,255 26x26), input disabled if: NOT fbMachine.bTestOutput, image: VisuSymbols.Symbols.Bracket
        OnMouseClick:  ToggleVariable=stFixInOuts.stBalluff.bDO_Trigger
    Image (294,285 26x26), input disabled if: NOT fbMachine.bTestOutput, image: VisuSymbols.Symbols.Bracket
        OnMouseClick:  ToggleVariable=stFixInOuts.bVacuumON_Q
END_VISUALIZATION

// ProdLineMachines/Sonictech/Fixtures/S01_IndicatorAssembly/VISUs/SubFrame/vStFix_S01IndicatorAssy_SubSettings
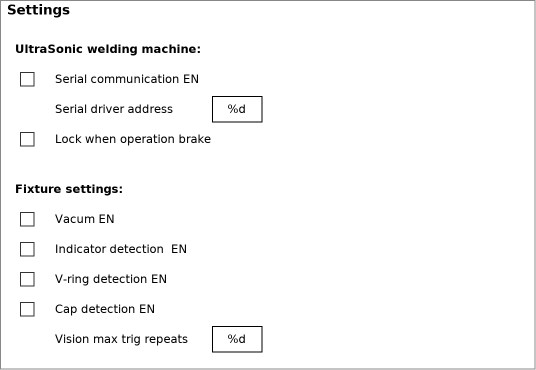
VISUALIZATION vStFix_S01IndicatorAssy_SubSettings  // 536x370
VAR_IN_OUT
	stSettings: stStFix_S01IndicatorAssy_Settings;
END_VAR
    Frame (0,0 536x370)
        shows vSonictechUSWM_SubSettings(stMachSettings := stSettings)
    Label (12,176 203x26), "Fixture settings:"
    Rectangle (52,206 160x26), "Vacum EN"
    Checkbox (18,206 26x26), variable: stSettings.bVacumEN
    Checkbox (18,236 26x26), variable: stSettings.bIndicatorCheckEN
    Rectangle (52,236 160x26), "Indicator detection EN"
    Checkbox (18,266 26x26), variable: stSettings.bVRingCheckEN
    Rectangle (52,266 160x26), "V-ring detection EN"
    Rectangle (52,296 160x26), "Cap detection EN"
    Checkbox (18,296 26x26), variable: stSettings.bCapCheckEN
    Rectangle (212,326 50x26), "%d", text variable: stSettings.iMaxTrigRepeats
        OnMouseClick: write the text variable via Default, min 0, max 5, title "Trig repeats"
    Rectangle (52,326 160x26), "Vision max trig repeats"
END_VISUALIZATION

// ProdLineMachines/Sonictech/Fixtures/S01_IndicatorAssembly/VISUs/vStFix_S01IndicatorAssy_Main
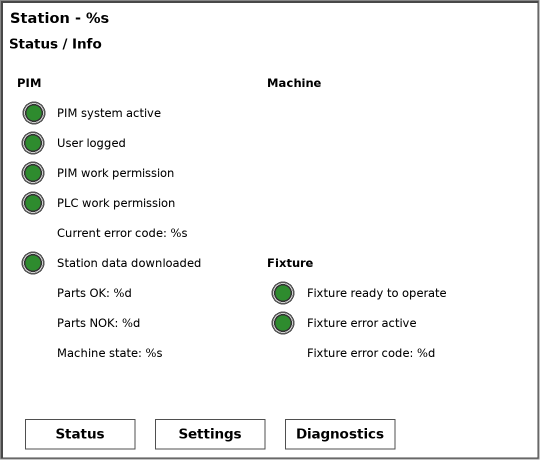
VISUALIZATION vStFix_S01IndicatorAssy_Main  // 540x460
VAR_IN_OUT
	fbPIM: fbPIM_Station_V3;
	fbMachine: fbSonictechUSWM;
	stSettings: stStFix_S01IndicatorAssy_Settings;
	stFixIO: stStFix_S01IndicatorAssy_InOut;
END_VAR
    Rectangle (1,1 538x458)
    Rectangle (25,419 110x30), "Status"
        OnMouseClick: FrameSelectionChange Selection=SelectedFrame=57fd262e-2fea-4fde-aa72-b89d7183eaaf, GlobSel=AssignType=Expression, SelType=Locally
        OnMouseClick: execute {  }
    Rectangle (155,419 110x30), "Settings"
        OnMouseClick: FrameSelectionChange Selection=SelectedFrame=57fd262e-2fea-4fde-aa72-b89d7183eaaf, Selection=1, GlobSel=AssignType=Expression, SelType=Locally
    Rectangle (285,419 110x30), "Diagnostics"
        OnMouseClick: FrameSelectionChange Selection=SelectedFrame=57fd262e-2fea-4fde-aa72-b89d7183eaaf, Selection=2, GlobSel=AssignType=Expression, SelType=Locally
    Rectangle (7,3 530x30), "Station - %s", text variable: fbPIM.sStationAlias
    Frame (2,34 536x370)
        shows vSonictechUSWM_SubStatus(fbMachine := fbMachine, fbPIM := fbPIM)
        shows vStFix_S01IndicatorAssy_SubSettings(stSettings := stSettings)
        shows vStFix_S01IndicatorAssy_SubDiag(fbMachine := fbMachine, stFixInOuts := stFixIO)
END_VISUALIZATION

// ProdLineMachines/Sonictech/Welding Machine/VISUs/SubFrame/vSonictechUSWM_SubDiag
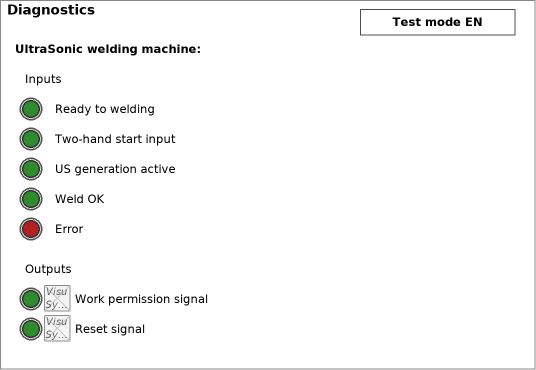
VISUALIZATION vSonictechUSWM_SubDiag  // 536x370
VAR_IN_OUT
	fbMachine: fbSonictechUSWM;
END_VAR
    Label (4,0 150x20), "Diagnostics"
    Label (12,36 203x26), "UltraSonic welding machine:"
    Lamp1 (18,96 26x26), variable: fbMachine.stDigitalInOut.bReadyToWelding, style: Lamp-Lamp1-Green
    Rectangle (52,96 160x26), "Ready to welding"
    Rectangle (52,126 160x26), "Two-hand start input"
    Lamp1 (18,126 26x26), variable: fbMachine.stDigitalInOut.bStartInput, style: Lamp-Lamp1-Green
    Lamp1 (18,156 26x26), variable: fbMachine.stDigitalInOut.bWeldingActive, style: Lamp-Lamp1-Green
    Rectangle (52,156 160x26), "US generation active"
    Rectangle (52,186 160x26), "Weld OK"
    Lamp1 (18,186 26x26), variable: fbMachine.stDigitalInOut.bWeld_OK, style: Lamp-Lamp1-Green
    Lamp1 (18,216 26x26), variable: fbMachine.stDigitalInOut.bErrorActive, style: Lamp-Lamp1-Red
    Rectangle (52,216 160x26), "Error"
    Rectangle (22,66 160x26), "Inputs"
    Rectangle (22,256 160x26), "Outputs"
    Lamp1 (18,316 26x26), variable: fbMachine.stDigitalInOut.bResetError, style: Lamp-Lamp1-Green
    Lamp1 (18,286 26x26), variable: fbMachine.stDigitalInOut.bWorkPermit, style: Lamp-Lamp1-Green
    Rectangle (72,286 150x26), "Work permission signal"
    Rectangle (72,316 150x26), "Reset signal"
    Rectangle (360,9 155x26), "Test mode EN", colour toggle: fbMachine.bTestOutput
        toggle fbMachine.bTestOutput
    Image (44,285 26x26), input disabled if: NOT fbMachine.bTestOutput, image: VisuSymbols.Symbols.Bracket
        OnMouseClick:  ToggleVariable=fbMachine.stDigitalInOut.bWorkPermit
    Image (44,315 26x26), input disabled if: NOT fbMachine.bTestOutput, image: VisuSymbols.Symbols.Bracket
        OnMouseClick:  ToggleVariable=fbMachine.stDigitalInOut.bResetError
END_VISUALIZATION

// ProdLineMachines/Sonictech/Welding Machine/VISUs/SubFrame/vSonictechUSWM_SubSettings
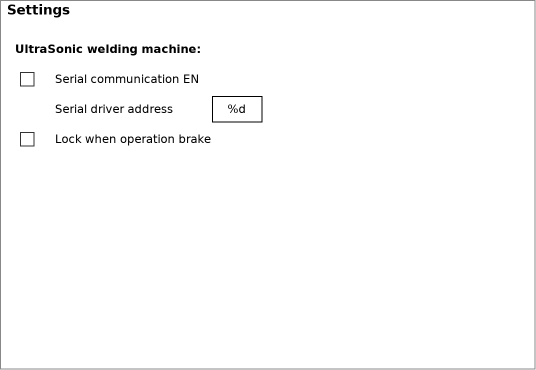
VISUALIZATION vSonictechUSWM_SubSettings  // 536x370
VAR_IN_OUT
	stMachSettings: stSonicTech_MachSettings;
END_VAR
    Label (4,0 150x20), "Settings"
    Label (12,36 245x26), "UltraSonic welding machine:"
    Rectangle (52,126 160x26), "Lock when operation brake"
    Rectangle (52,66 160x26), "Serial communication EN"
    Checkbox (18,66 26x26), variable: stMachSettings.bSerialCommunicationEN
    Checkbox (18,126 26x26), variable: stMachSettings.bLockWhenOperationsBreaked
    Rectangle (212,96 50x26), "%d", text variable: stMachSettings.bySerialAdress
        OnMouseClick: write the text variable via Default, min 0, max 126, title "Serial address"
    Rectangle (52,96 160x26), "Serial driver address"
END_VISUALIZATION

// ProdLineMachines/Sonictech/Welding Machine/VISUs/SubFrame/vSonictechUSWM_SubStatus
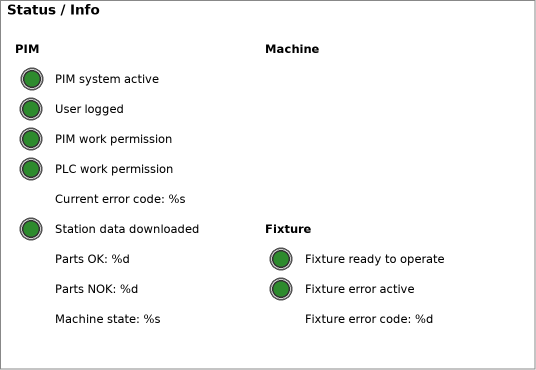
VISUALIZATION vSonictechUSWM_SubStatus  // 536x370
VAR_IN_OUT
	fbMachine: fbSonictechUSWM;
	fbPIM: fbPIM_Station_V3;
END_VAR
    Label (4,0 150x20), "Status / Info"
    Label (12,36 150x26), "PIM"
    Rectangle (52,96 160x26), "User logged"
    Rectangle (52,126 160x26), "PIM work permission"
    Rectangle (52,156 160x26), "PLC work permission"
    Rectangle (52,216 160x26), "Station data downloaded"
    Rectangle (52,246 160x26), "Parts OK: %d"
    Rectangle (52,276 160x26), "Parts NOK: %d"
    Rectangle (52,306 200x26), "Machine state: %s", text variable: TO_STRING(fbPIM.nMachineState)
    Label (262,36 150x26), "Machine"
    Rectangle (52,66 160x26), "PIM system active"
    Label (262,216 150x26), "Fixture", invisible if: NOT fbMachine.bFixConnected
    Lamp1 (268,246 26x26), variable: fbMachine.bFixtureReady, invisible if: NOT fbMachine.bFixConnected, style: Lamp-Lamp1-Green
    Rectangle (302,246 160x26), "Fixture ready to operate", invisible if: NOT fbMachine.bFixConnected
    Lamp1 (268,276 26x26), variable: fbMachine.bFixError, invisible if: NOT fbMachine.bFixConnected, style: Lamp-Lamp1-Green
    Rectangle (302,276 160x26), "Fixture error active", invisible if: NOT fbMachine.bFixConnected
    Rectangle (302,306 160x26), "Fixture error code: %d", text variable: fbMachine.iFixErrorCode, invisible if: NOT fbMachine.bFixConnected
    Lamp1 (19,66 26x26), variable: fbPIM.stPimInOut.bPIMActive, style: Lamp-Lamp1-Green
    Lamp1 (18,96 26x26), variable: fbPIM.stPimInOut.bUserLogged, style: Lamp-Lamp1-Green
    Lamp1 (18,126 26x26), variable: NOT fbPIM.stPimInOut.bWorkBlock_PIM, style: Lamp-Lamp1-Green
    Lamp1 (18,156 26x26), variable: NOT fbPIM.stPimInOut.bWorkBlock_PLC, style: Lamp-Lamp1-Green
    Rectangle (52,186 160x26), "Current error code: %s", text variable: fbPIM.stPimInOut.sErrorCodePLC
    Lamp1 (18,216 26x26), variable: fbPIM.bStationDataOK, style: Lamp-Lamp1-Green
END_VISUALIZATION

// ProdLineMachines/Sonictech/Welding Machine/VISUs/vSonictechUSWM_Main
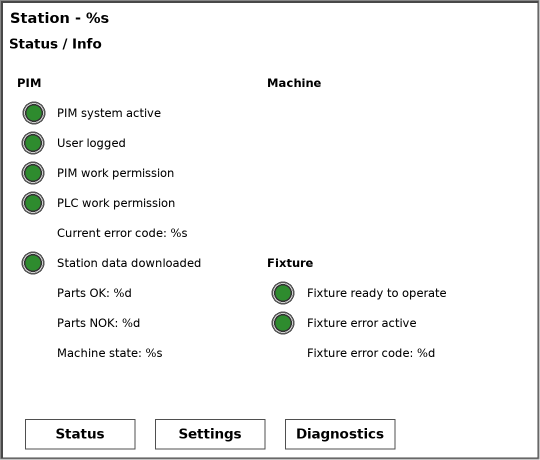
VISUALIZATION vSonictechUSWM_Main  // 540x460
VAR_IN_OUT
	fbPIM: fbPIM_Station_V3;
	fbMachine: fbSonictechUSWM;
	stMachSettings: stSonicTech_MachSettings;
END_VAR
    Rectangle (1,1 538x458)
    Rectangle (25,419 110x30), "Status"
        OnMouseClick: FrameSelectionChange Selection=SelectedFrame=57fd262e-2fea-4fde-aa72-b89d7183eaaf, GlobSel=AssignType=Expression, SelType=Locally
        OnMouseClick: execute { fbMachine.bTestOutput:= FALSE; }
    Rectangle (155,419 110x30), "Settings"
        OnMouseClick: FrameSelectionChange Selection=SelectedFrame=57fd262e-2fea-4fde-aa72-b89d7183eaaf, Selection=1, GlobSel=AssignType=Expression, SelType=Locally
        OnMouseClick: execute { fbMachine.bTestOutput:= FALSE; }
    Rectangle (285,419 110x30), "Diagnostics"
        OnMouseClick: FrameSelectionChange Selection=SelectedFrame=57fd262e-2fea-4fde-aa72-b89d7183eaaf, Selection=2, GlobSel=AssignType=Expression, SelType=Locally
    Frame (2,34 536x370)
        shows vSonictechUSWM_SubStatus(fbMachine := fbMachine, fbPIM := fbPIM)
        shows vSonictechUSWM_SubSettings(stMachSettings := stMachSettings)
        shows vSonictechUSWM_SubDiag(fbMachine := fbMachine)
    Rectangle (7,3 530x30), "Station - %s", text variable: fbPIM.sStationAlias
END_VISUALIZATION

// SQL/VISUs/vSQL_Core_AlarmTab
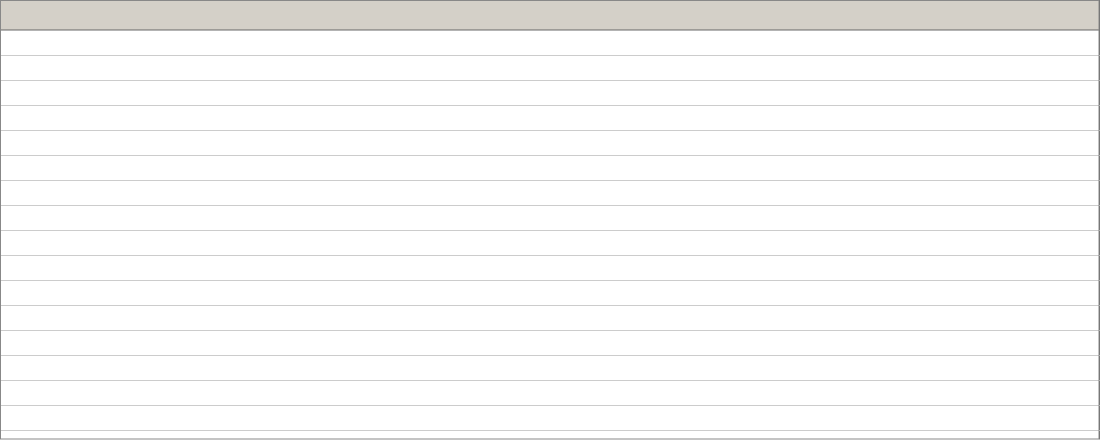
VISUALIZATION vSQL_Core_AlarmTab  // 1100x440
VAR_IN_OUT
	fbData:fbAlarmSlaveTable;
END_VAR
    Table (0,0 1100x439), data array: fbData.astErrTable
        p3854506369: fbData.astErrTable[INDEX].dtEventTime
        p1892666644: fbData.astErrTable[INDEX].sMachineId
        p338671338: fbData.astErrTable[INDEX].sEventDescription
        p2170511999: fbData.astErrTable[INDEX].dwErrorCode
        p3723444502: fbData.astErrTable[INDEX].uiRepeatQty
        p1218418051: fbData.astErrTable[INDEX].nAlarmClass
        p2232123230: Event Time
        p1755163831: Event Description
        p4092479075: Error Code
        p2237128397: Repeat Qty
        p1128707560: fbData.uiRowNumber
END_VISUALIZATION

// SQL/VISUs/vSQL_CoreDiag
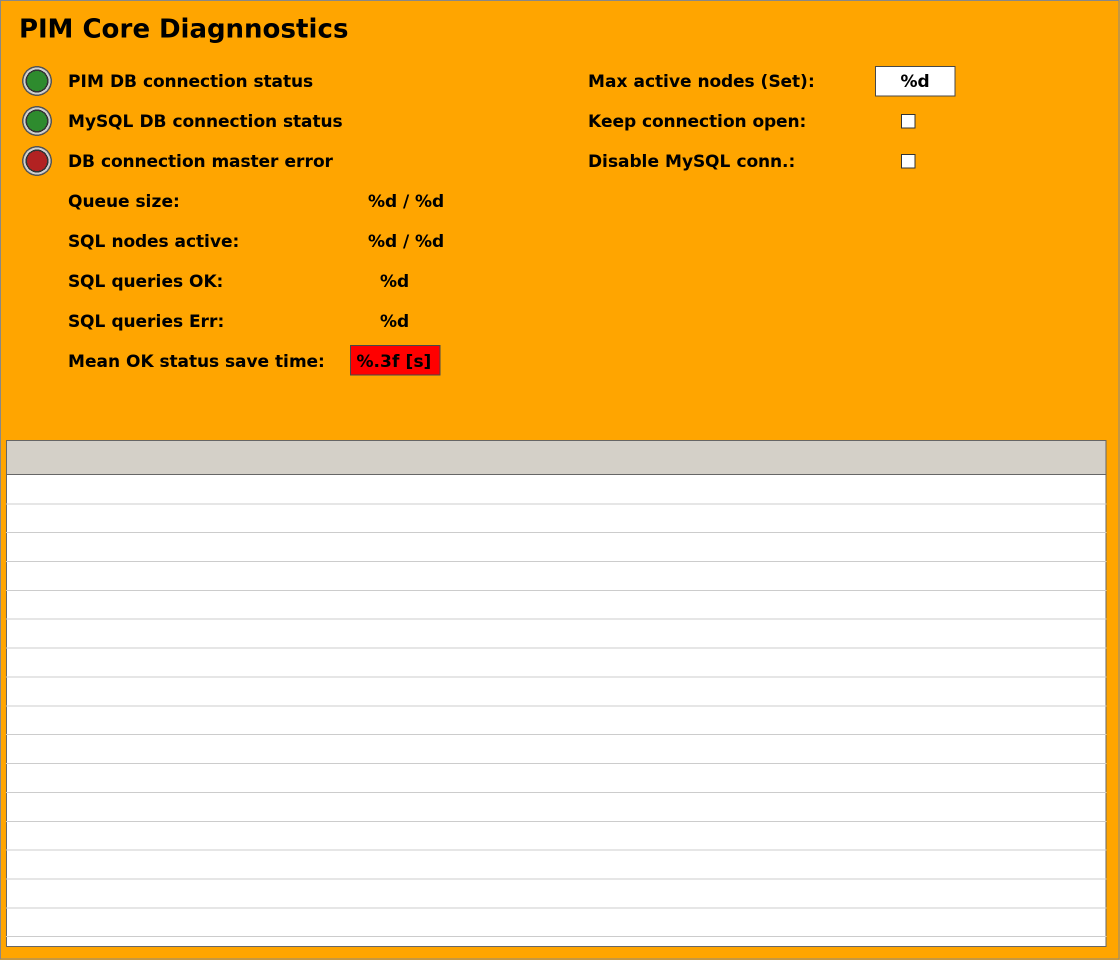
VISUALIZATION vSQL_CoreDiag  // 1120x960
VAR_IN_OUT
	fbData: fbSQL_Core;
END_VAR
    Rectangle (16,11 375x43), "PIM Core Diagnnostics"
    Lamp1 (20,64 34x34), variable: fbData.bConnectionMSSQL_OK, style: Lamp-Lamp1-Green
    Rectangle (65,66 300x30), "PIM DB connection status"
    Lamp1 (20,144 34x34), variable: fbData.bMasterError, style: Lamp-Lamp1-Red
    Rectangle (65,146 300x30), "DB connection master error"
    Label (65,186 280x30), "Queue size:"
    Rectangle (337,186 63x30), "%d", text variable: fbData.iQueueLastCmdIndex
    Lamp1 (20,104 34x34), variable: fbData.bConnectionMySQL_OK, style: Lamp-Lamp1-Green
    Rectangle (65,106 300x30), "MySQL DB connection status"
    Rectangle (400,186 63x30), "/ %d", text variable: fbData.iQueueSize
    Label (65,226 280x30), "SQL nodes active:"
    Rectangle (337,226 63x30), "%d", text variable: fbData.iActiveNodesNb
    Rectangle (400,226 63x30), "/ %d", text variable: fbData.iMaxActiveNodesNb
    Rectangle (363,306 63x30), "%d", text variable: fbData.udiSQL_Queries_ERR
    Rectangle (363,266 63x30), "%d", text variable: fbData.udiSQL_Queries_OK
    Rectangle (350,345 90x30), invisible if: NOT fbData.fbFilter_Warning.Q
    Label (65,266 280x30), "SQL queries OK:"
    Label (65,306 280x30), "SQL queries Err:"
    Label (65,346 280x30), "Mean OK status save time:"
    Rectangle (875,66 80x30), "%d", text variable: fbData.iMaxActiveNodesNb, input disabled if: Not GVL_Aircom.bPermissionGranted
        OnMouseClick: write the text variable via Default, min 3, max 8
    Label (585,66 290x30), "Max active nodes (Set):"
    Label (585,106 290x30), "Keep connection open:"
    Checkbox (899,106 30x30), variable: fbData.bKeepConnOpen, input disabled if: Not GVL_Aircom.bPermissionGranted
    Label (585,146 290x30), "Disable MySQL conn.:"
    Checkbox (899,146 30x30), variable: fbData.bDisableMySQL, input disabled if: Not GVL_Aircom.bPermissionGranted
    Rectangle (350,345 90x30), invisible if: NOT fbData.fbFilter_Alarm.Q
    Rectangle (349,346 90x30), "%.3f [s]", text variable: fbData.rMeanOkCmdTime
    Frame (6,440 1100x508)
        shows vSQL_Core_AlarmTab(fbData := fbData.fbAlarmTab)
END_VISUALIZATION
